(* PLC project addition, Dassault Systèmes ControlBuild 2024x *)
(* stored: creationDateTime 2023-10-03T11:13:25-01:00 *)

(* This module simulates the addition of two real numbers. *)
FUNCTION_BLOCK equipment_library.addition
  VAR_INPUT
    in1 : REAL := 0.0;
    in2 : REAL := 0.0;
  END_VAR
  VAR_OUTPUT
    value : REAL := 0.0;
    dintValue : DINT := 0;
    intValue : INT := 0;
  END_VAR
  VAR
    d_locking : BOOL := false;
    v_d_locking : REAL := 0.0;
  END_VAR


ACTION C_source_code:
/* ----------------------------------------------------------------	*/
/* Type : Model of Operative Behaviour					*/
/* Category :  Toolbox							*/
/* Author : Dassault Systemes						*/
/* Update date : June 2018						*/
/* ----------------------------------------------------------------	*/
/* This module simulates the addition of two real numbers.		*/
/* ----------------------------------------------------------------	*/

if (d_locking)
	value = v_d_locking;	 /* presetting of the value */
else
	value = in1+in2;		 /* addition result		 */

dintValue = value;

if ((dintValue >= -32768) && (dintValue <= 32767)) 
	intValue = dintValue ;
else 
	intValue  = 0;
END_ACTION
END_FUNCTION_BLOCK
